(* PLC project Transportband_ohne_Trans, KW-Software MULTIPROG 5.35 *)
(* stored: companyURL www.kw-software.com, productRelease Build 434, creationDateTime 2012-11-09T12:51:59, version 1352461919, modificationDateTime 2012-11-09T12:51:59 *)

(* Layer 3: Ablaufebene (Version 2: 1 Sensor mittig) --> Greift auf Layer 2 zu. Der FB spiegelt die Funktion "Transport nach x" eines Werkstücks wider. Der Unterschied zum FB "Transportieren" aus Layer 2 besteht darin, dass der Transportablauf neben dem reinen Transportieren auch die Übernahme und Übergabe des Werkstücks umfasst. Die Ansteuerung der drei Transportierenzustände (links, rechts, aus) wird durch zwei Transportrichtungsvariablen (links und rechts) realisiert. Im Anfangsschritt findet kein Transportablauuf statt - kein Transportieren/Übergeben/Übernehmen (Motoren aus). Je nach Setzen der Inputvariablen (alternative Verzweigung) wird nach links oder rechts transportiert - die Transition "T_xxx_ein" schaltet. Dadurch wird der Zustand eingenommen, in dem ein Werkstück von der entsprechenden Seite übernommen wird. Liefert FB "Übernahme_gabe" das Quittierungssignal, dass erfolgreich übernommen wurde, schaltet die Transition. Damit wird der Transportieren-Zustand eingenommen. Wurde erfolgreich transportiert und somit das Qittierungssignal des FB zurückgegeben, so schaltet die Transition und es wird der Folgzustand eingenommen - Übergeben. Wurde erfolgreich übergeben, so ist der Transportablauf abgeschlossen. Dabei wird auch eine Statusvariable gesetzt (TPx_xxx), die den erfolgreichen Transportablauf quittiert, sodass die übergeordnete Steuerung weiß, wann der Transportvorgang abgeschlossen ist. FB-Schnittstellen: --------------- Eingangsvariablen: - Transport_nach_links - Transport_nach_rechts Ausgangsvariablen: - TPx_links - TPx_rechts Auftretende Warnungen "Instanz 'FB_xxx' mehrfach verwendet!": Hier ein Textauszug aus der Multiprog-Hilfe: "Die Warnung kann auch in einem Code-Arbeitsblatt in AS auftreten, wenn Sie dieselbe Instanz in verschiedenen Aktionen verwendet haben. Wenn nur eine Instanz zu einem Zeitpunkt ausgeführt wird, ist die Warnung für Sie ohne Bedeutung." *)
FUNCTION_BLOCK Transport_zu_x
  VAR_INPUT
    Transport_nach_links : BOOL := FALSE;  (* Inputvariable *)
    Transport_nach_rechts : BOOL := FALSE;  (* Inputvariable *)
  END_VAR
  VAR
    FB_Uebergabe : Uebernahme_gabe;  (* Outputvariable vom FB "Uebernahme_gabe". Quittierungssignal für Übergabe *)
    Quittierungssignal_links1 : BOOL := FALSE;  (* Hilfsvariable: Hier wird der Output des Uebergabe/Transportieren-FBs eingetragen. Es wurde nach links übergeben. ODER es wurde nach links transportiert. *)
    Quittierungssignal_rechts1 : BOOL := FALSE;  (* Hilfsvariabel: Hier wird der Output des Uebergabe/Transportieren-FBs eingetragen. Es wurde nach rechts übergeben. ODER es wurde nach rechts transportiert. *)
  END_VAR
  VAR_OUTPUT
    TPx_links : BOOL := FALSE;  (* Quittierungssignal: Es wurde nach links transportiert. *)
    TPx_rechts : BOOL := FALSE;  (* Quittierungssignal: Es wurde nach rechts transportiert, *)
  END_VAR
  VAR
    Quittierungssignal_links2 : BOOL := FALSE;
    Quittierungssignal_rechts2 : BOOL := FALSE;
    Quittierungssignal_links3 : BOOL := FALSE;
    Quittierungssignal_rechts3 : BOOL := FALSE;
    FB_Uebernahme : Uebernahme_gabe;  (* Outputvariable vom FB "Uebernahme_gabe". Quittierungssignal für Übernahme *)
  END_VAR

(* transition T_Uebernehmen_l_ein *)
(*Wird vom Anwender oder vom darüberliegenden Layer die Entscheidung getroffen, dass das Transportband nach links befördern soll, 
dann wird die Transition gesetzt und der Folgezustand wird eingenommen.*)
IF Transport_nach_links = TRUE AND Transport_nach_rechts = FALSE
	THEN T_Uebernehmen_l_ein := TRUE;
	ELSE T_Uebernehmen_l_ein := FALSE;
END_IF;
(* transition T_Transportablauf_l_aus *)
(*Statusvariablenabfrage.*)

(*Der FB "Übernahme_gabe" aus Layer 2 wird jeweils für Linksbewegung instanziiert.*)
FB_Uebergabe();

(*Der lokalen (Hilfs-)Variable "Quittierungssignal_links" wird der jeweilige Ausgangwert des FBs "Übernahme_gabe" zugewiesen.*)
Quittierungssignal_links3 := FB_Uebergabe.UeG_UeN_links;

(*Wenn das Quittierungssignal TRUE ist, gilt das Werkstück als erfolgreich übergeben und die Transition wird gesetzt.*)
IF Quittierungssignal_links3 = TRUE
	THEN T_Transportablauf_l_aus := TRUE;
	ELSE T_Transportablauf_l_aus := FALSE;
END_IF;
(* transition T_Uebernehmen_r_ein *)
(*Wird vom Anwender oder vom darüberliegenden Layer die Entscheidung getroffen, dass das Transportband nach rechts befördern soll, 
dann wird die Transition gesetzt und der Folgezustand wird eingenommen.*)
IF Transport_nach_rechts = TRUE AND Transport_nach_links = FALSE
	THEN T_Uebernehmen_r_ein := TRUE;
	ELSE T_Uebernehmen_r_ein := FALSE;
END_IF;
(* transition T_Transportablauf_r_aus *)
(*Statusvariablenabfrage.*)

(*Der FB "Übernahme_gabe" aus Layer 2 wird jeweils für Rechtsbewegung instanziiert.*)
FB_Uebergabe();

(*Der lokalen (Hilfs-)Variable "Quittierungssignal_links" wird der jeweilige Ausgangwert des FBs "Übernahme_gabe" zugewiesen.*)
Quittierungssignal_rechts3 := FB_Uebergabe.UeG_UeN_rechts;

(*Wenn das Quittierungssignal TRUE ist, gilt das Werkstück als erfolgreich übergeben und die Transition wird gesetzt.*)
IF Quittierungssignal_rechts3 = TRUE 
	THEN T_Transportablauf_r_aus := TRUE;
	ELSE T_Transportablauf_r_aus := FALSE;
END_IF;
(* transition T_Uebergeben_l_ein *)
(*Statusvariablenabfrage.*)

FB_Uebernahme();

Quittierungssignal_links2 := FB_Uebernahme.UeG_UeN_links;

(*Wenn das Quittierungssignal TRUE ist, gilt das Werkstück als erfolgreich transportiert und die Transition wird gesetzt.*)
IF Quittierungssignal_links2 = TRUE
	THEN T_Uebergeben_l_ein := TRUE;
	ELSE T_Uebergeben_l_ein := FALSE;
END_IF;
(* transition T_Uebergeben_r_ein *)
(*Statusvariablenabfrage.*)

FB_Uebernahme();

Quittierungssignal_rechts2 := FB_Uebernahme.UeG_UeN_rechts;

(*Wenn das Quittierungssignal TRUE ist, gilt das Werkstück als erfolgreich transportiert und die Transition wird gesetzt.*)
IF Quittierungssignal_rechts2 = TRUE 
	THEN T_Uebergeben_r_ein := TRUE;
	ELSE T_Uebergeben_r_ein := FALSE;
END_IF;
(* transition T_sofort_weiter5 *)
(*In dieser Transition steckt keine Bedingung. Die Transition wird sofort gesetzt und der Folgezustand wird eingenommen.*)
(* transition T_sofort_weiter6 *)
(*In dieser Transition steckt keine Bedingung. Die Transition wird sofort gesetzt und der Folgezustand wird eingenommen.*)
INITIAL_STEP Motor_aus:
END_STEP
TRANSITION FROM Motor_aus TO Motor_links_UeN
  := T_Uebernehmen_l_ein;
END_TRANSITION
TRANSITION FROM Motor_aus TO Motor_rechts_UeN
  := T_Uebernehmen_r_ein;
END_TRANSITION
STEP Motor_links_UeN:
END_STEP
TRANSITION FROM Motor_links_UeN TO Motor_links_UeG
  := T_Uebergeben_l_ein;
END_TRANSITION
STEP Motor_rechts_UeN:
END_STEP
TRANSITION FROM Motor_rechts_UeN TO Motor_rechts_UeG
  := T_Uebergeben_r_ein;
END_TRANSITION
STEP Motor_links_UeG:
END_STEP
TRANSITION FROM Motor_links_UeG TO Quittierung_l
  := T_Transportablauf_l_aus;
END_TRANSITION
STEP Motor_rechts_UeG:
END_STEP
TRANSITION FROM Motor_rechts_UeG TO Quittierung_r
  := T_Transportablauf_r_aus;
END_TRANSITION
STEP Quittierung_l:
END_STEP
TRANSITION FROM Quittierung_l TO Endschritt_3  (* T_sofort_weiter5 *)
  := TRUE;
END_TRANSITION
STEP Quittierung_r:
END_STEP
TRANSITION FROM Quittierung_r TO Endschritt_3  (* T_sofort_weiter6 *)
  := TRUE;
END_TRANSITION
STEP Endschritt_3:
END_STEP

ACTION Uebernehmen_von_links:
(*In diesem Zustand befindet sich der Motor in der Rechtsdrehung - Werkstück wird übernommen.
Layer 3 greift auch Layer 2 "Übernahme_gabe" zu und setzt die Eingangsvariablen dieses FBs entsprechend.*)

(*von links übernehmen*)
FB_Uebernahme(Richtung := FALSE, Uebernehmen := TRUE, Uebergeben := FALSE);
END_ACTION

ACTION Uebernehmen_von_rechts:
(*In diesem Zustand befindet sich der Motor in der Linksdrehung - Werkstück wird übernommen.
Layer 3 greift auch Layer 2 "Übernahme_gabe" zu und setzt die Eingangsvariablen dieses FBs entsprechend.*)

(*von rechts übernehmen*)
FB_Uebernahme(Richtung := TRUE, Uebernehmen := TRUE, Uebergeben := FALSE);
END_ACTION

ACTION Uebergeben_nach_links:
(*In diesem Zustand befindet sich der Motor in der Linksdrehung - Werkstück wird übergeben.
Layer 3 greift auch Layer 2 "Übernahme_gabe" zu und setzt die Eingangsvariablen dieses FBs entsprechend.*)

(*nach links übergeben*)
FB_Uebergabe(Richtung := FALSE, Uebernehmen := FALSE, Uebergeben := TRUE);
END_ACTION

ACTION Uebergeben_nach_rechts:
(*In diesem Zustand befindet sich der Motor in der Rechtsdrehung - Werkstück wird übergeben.
Layer 3 greift auch Layer 2 "Übernahme_gabe" zu und setzt die Eingangsvariablen dieses FBs entsprechend.*)

(*nach rechts übergeben*)
FB_Uebergabe(Richtung := TRUE, Uebernehmen := FALSE, Uebergeben := TRUE);
END_ACTION

ACTION Quittierung_links3:
(*Statusvariable: Wird gesetzt, wenn bei Linksdrehung erfolgreich der Transportablauf erledigt wurde.
Diese Signal ist nötig für übergeordnete Steuerungen.*)
TPx_links := TRUE;
END_ACTION

ACTION Quittierung_rechts3:
(*Statusvariable: Wird gesetzt, wenn bei Rechtsdrehung erfolgreich der Transportablauf erledigt wurde.
Diese Signal ist nötig für übergeordnete Steuerungen.*)
TPx_rechts := TRUE;
END_ACTION

ACTION Transportablauf_aus:
(*In diesem Zustand befindet sich der Motor im unbestromten Zustand - Also kein Transportieren/Übergeben/Übernehmen.
Layer 3 greift auch Layer 2 "Transportieren" und "Übernahme_gabe" zu und setzt die Eingangsvariablen dieser FBs entsprechend.*)

FB_Uebernahme(Uebergeben := FALSE, Uebernehmen := FALSE);
FB_Uebergabe(Uebergeben := FALSE, Uebernehmen := FALSE);
END_ACTION

ACTION Endschritt_Ablauf:
(*In diesem Zustand befindet sich der Motor im unbestromten Zustand - Also kein Transportieren/Übergeben/Übernehmen.
Layer 3 greift auch Layer 2 "Transportieren" und "Übernahme_gabe" zu und setzt die Eingangsvariablen dieser FBs entsprechend.*)
FB_Uebernahme(Uebergeben := FALSE, Uebernehmen := FALSE);
FB_Uebergabe(Uebergeben := FALSE, Uebernehmen := FALSE);
END_ACTION
END_FUNCTION_BLOCK
